(* Schneider Machine Expert - Basic project Multiple Motor Connections, file version 2.9.0.0 *)
(* ProjectInformations: Name=New project *)

HARDWARE
  Cpu 0: TM221C24R
  EthernetConfiguration: NetworkName=M221, IpAllocationMode=FixedAddress, IpAddress=0.0.0.0, SubnetMask=0.0.0.0
  SerialLineConfiguration: Baud=Baud19200, Parity=ParityEven, DataBits=DataBits8, StopBits=StopBits1, PhysicalMedium=PhysicalMediumRs485, SlaveId=1, Addressing=SlaveAddressing
  MastTask: UsePeriodScanMode=false, PeriodScan=100
  FastTask: Period=255
  CpuBehavior: StartingMode=StartAsPreviousState, AutoSaveRamOnEeprom=true, WatchdogPeriod=250

SYMBOLS  (address, symbol, comment, settings)
  %I0.0     SWITCH_1
  %I0.1     SWITCH_2
  %I0.2     SWITCH_3
  %Q0.0     MOTOR_1
  %Q0.1     MOTOR_2
  %Q0.2     MOTOR_3

POU New POU
  (* SectionNumber=1 *)

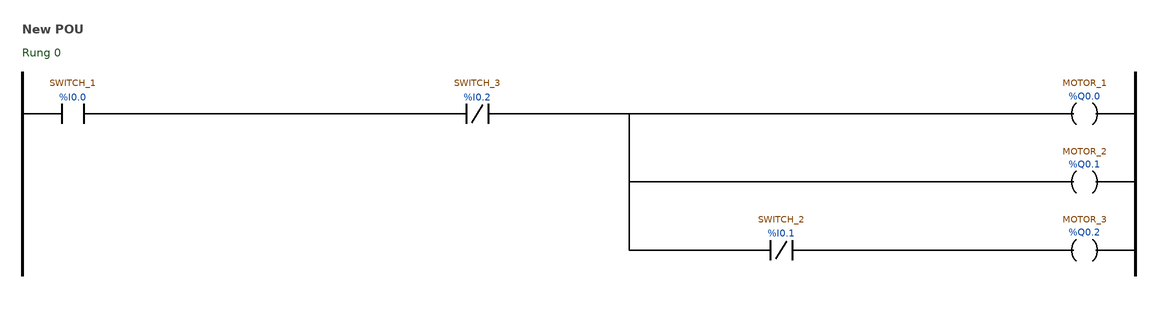

// Rung 0
  LD %I0.0                (* SWITCH_1 *)
  ANDN %I0.2              (* SWITCH_3 *)
  MPS
  ST %Q0.0                (* MOTOR_1 *)
  MRD
  ST %Q0.1                (* MOTOR_2 *)
  MPP
  ANDN %I0.1              (* SWITCH_2 *)
  ST %Q0.2                (* MOTOR_3 *)
  // as ST:
  //   MOTOR_1 := SWITCH_1 AND NOT SWITCH_3;
  //   MOTOR_2 := SWITCH_1 AND NOT SWITCH_3;
  //   MOTOR_3 := SWITCH_1 AND NOT SWITCH_3 AND NOT SWITCH_2;
